DATA_BLOCK "ST10_Stopper_FB_DB"
{ S7_Optimized_Access := 'TRUE' }
VERSION : 0.1
NON_RETAIN
"ST10_Stopper_FB"

BEGIN

END_DATA_BLOCK

